FUNCTION_BLOCK FB_HE_SATT_EpicsHeartBeatTest EXTENDS FB_TestSuite


GivenThatHeartbeatIsProvidedExpectNoExpiration();
GivenThatHeartbeatTimeHasExpiredExpectHeartBeatPropertyToIndicateSo();


METHOD PRIVATE GivenThatHeartbeatIsProvidedExpectNoExpiration
VAR_INST
    fbTestTimer : TON := (PT := T#2S, IN := TRUE);

    // Subject under test
    fbHE_SATT_EpicsHeartBeat : FB_HE_SATT_EpicsHeartBeat(tTimeout := T#1S);
END_VAR

TEST('GivenThatHeartbeatIsProvidedExpectNoExpiration');

fbTestTimer();
fbHE_SATT_EpicsHeartBeat.Heartbeat();
fbHE_SATT_EpicsHeartBeat();

IF fbTestTimer.Q THEN
    AssertFalse(Condition := fbHE_SATT_EpicsHeartBeat.IsHeartbeatExpired(),
                Message := 'Expected heart beat to expire');
    TEST_FINISHED();
END_IF
END_METHOD


METHOD PRIVATE GivenThatHeartbeatTimeHasExpiredExpectHeartBeatPropertyToIndicateSo
VAR_INST
    fbTestTimer : TON := (PT := T#2S, IN := TRUE);

    // Subject under test
    fbHE_SATT_EpicsHeartBeat : FB_HE_SATT_EpicsHeartBeat(tTimeout := T#1S);
END_VAR

TEST('GivenThatHeartbeatTimeHasExpiredExpectHeartBeatPropertyToIndicateSo');

fbTestTimer();
fbHE_SATT_EpicsHeartBeat();

IF fbTestTimer.Q THEN
    AssertTrue(Condition := fbHE_SATT_EpicsHeartBeat.IsHeartbeatExpired(),
               Message := 'Expected heart beat to expire');
    TEST_FINISHED();
END_IF
END_METHOD

END_FUNCTION_BLOCK

(* stored: Version 1.1.0.1
   POU FB_HE_SATT_EpicsHeartBeatTest: Id {6737a63f-a220-4ec1-8820-e4e83f0e728d}, SpecialFunc None
   Method GivenThatHeartbeatIsProvidedExpectNoExpiration: Id {183df5e8-050c-41bd-b698-3a77bba84f8f}
   Method GivenThatHeartbeatTimeHasExpiredExpectHeartBeatPropertyToIndicateSo: Id {404e4665-6ffc-4dc9-aa69-d946929e3d31} *)
